INTERFACE I_Stop

PROPERTY PUBLIC Busy : BOOL
GET
END_GET
END_PROPERTY

PROPERTY PUBLIC Error : BOOL
GET
END_GET
END_PROPERTY

METHOD PUBLIC Parameterise : BOOL
VAR_INPUT
	deceleration : LREAL;
	jerk : LREAL;
END_VAR
END_METHOD

METHOD PUBLIC RegisterAxis : BOOL
VAR_IN_OUT
	axisRef : AXIS_REF;
END_VAR
END_METHOD

METHOD Stop
END_METHOD

END_INTERFACE

(* stored: Version 1.1.0.1, ProductVersion 3.1.4024.3
   Itf I_Stop: Id {abc908d2-d9b9-4dde-941b-d5a60f34d777}
   Property Busy: Id {3c3a6ca2-2e86-47cf-b238-66e572600910}
   Get Get: Id {fb6d93f4-e213-4df6-ae04-0752ba4e2ad2}
   Property Error: Id {ec1ba631-9a0d-4ec1-b754-9d3b39e965a9}
   Get Get: Id {ad070c08-7c7e-4eac-a0f4-7acc391f6427}
   Method Parameterise: Id {94ff68cb-71da-4757-aa18-2a29d121dd40}
   Method RegisterAxis: Id {44598adf-bba4-4a3a-bde9-522aefb1d52f}
   Method Stop: Id {a061b992-b6ea-479c-a64f-2105bfe9fff4} *)
